// Implicitly generated code : DO NOT EDIT
FUNCTION CheckDivLReal : LREAL
VAR_INPUT
	divisor:LREAL;
END_VAR

// Implicitly generated code : Only an Implementation suggestion
{noflow}
IF divisor = 0 THEN
	CheckDivLReal:=1;
ELSE
	CheckDivLReal:=divisor;
END_IF;
{flow}

END_FUNCTION

(* stored: Version 1.1.0.1, ProductVersion 3.1.4024.12
   POU CheckDivLReal: Id {a96703ad-56fb-4db1-b708-1f3f494f6cb6}, SpecialFunc CheckDivReal64 *)
